KUKA KRL program: machina_kuka_driver.src, machina_kuka_driver.dat

--- machina_kuka_driver.src ---
&ACCESS RVP
&REL 53
&PARAM DISKPATH = KRC:\R1\Program\Arastoo\Driver
&PARAM TEMPLATE = C:\KRC\Roboter\Template\vorgabe
&PARAM EDITMASK = *
DEF machina_kuka_driver( )

;FOLD INI
;FOLD BCO INI
GLOBAL INTERRUPT DECL 3 WHEN $STOPMESS==TRUE DO IR_STOPM ( )
INTERRUPT ON 3
BAS (#INITMOV,0 )
;ENDFOLD (BCO INI)
;ENDFOLD (INI)



; For KUKA 3 files need to be installed: .src driver, .dat data file, and .xml server configurations
; in the xml file we specify the precise format of each action, accessed by the src driver program
; This file starts a TCP server on a real KUKA robot,
; waits for a TCP client, listens to a stream of formatted string messages in xml,
; buffers them parsed into an 'action' struct, and runs a loop to execute them.

; IMPORTANT: make sure to adjust {{HOSTNAME}} and {{PORT}} to your current setup
; More info on https://github.com/RobotExMachina
; A project by https://github.com/garciadelcastillo

; MIT License

; Copyright (c) 2018 Jose Luis Garcia del Castillo y Lopez

; Permission is hereby granted, free of charge, to any person obtaining a copy
; of this software and associated documentation files (the "Software"), to deal
; in the Software without restriction, including without limitation the rights
; to use, copy, modify, merge, publish, distribute, sublicense, and/or sell
; copies of the Software, and to permit persons to whom the Software is
; furnished to do so, subject to the following conditions:

; The above copyright notice and this permission notice shall be included in all
; copies or substantial portions of the Software.

; THE SOFTWARE IS PROVIDED "AS IS", WITHOUT WARRANTY OF ANY KIND, EXPRESS OR
; IMPLIED, INCLUDING BUT NOT LIMITED TO THE WARRANTIES OF MERCHANTABILITY,
; FITNESS FOR A PARTICULAR PURPOSE AND NONINFRINGEMENT. IN NO EVENT SHALL THE
; AUTHORS OR COPYRIGHT HOLDERS BE LIABLE FOR ANY CLAIM, DAMAGES OR OTHER
; LIABILITY, WHETHER IN AN ACTION OF CONTRACT, TORT OR OTHERWISE, ARISING FROM,
; OUT OF OR IN CONNECTION WITH THE SOFTWARE OR THE USE OR OTHER DEALINGS IN THE
; SOFTWARE.

; specifying the robot will read 3 commands in advance so that it can blend movements
$ADVANCE=3

; Initializing a TCP server on the robot and listening for clients and messages
RET=EKI_Init("machina_kuka_server")
RET=EKI_Open("machina_kuka_server")

;PTP {A1 0,A2 -85,A3 105,A4 0,A5 -20,A6 0}
;FOLD INI
;FOLD BCO INI
GLOBAL INTERRUPT DECL 3 WHEN $STOPMESS==TRUE DO IR_STOPM ( )
INTERRUPT ON 3
BAS (#INITMOV,0 )
;ENDFOLD (BCO INI)
;ENDFOLD (INI)

; Setting status and turn for the initial position of the robot
; status and turn define the joint configuration of a robot for a position
joint_pos_tgt = $axis_act_meas
PTP joint_pos_tgt
current_position = $POS_ACT_MES
IK_pose_position = {X 0,Y 0,Z 0,A 0,B 0,C 0}
IK_pose_position.X = current_position.X
IK_pose_position.Y = current_position.Y
IK_pose_position.Z = current_position.Z
IK_pose_position.A = current_position.A
IK_pose_position.B = current_position.B
IK_pose_position.C = current_position.C
PTP IK_pose_position C_PTP
$TOOL = $NULLFRAME

$VEL.CP=0.02
FOR FI=1 TO 6
$VEL_AXIS[FI] = 10 ;all axis velocities to 10%
ENDFOR

; setting default movement path blending values
$APO.CDIS = 5
$APO.CPTP = 5

wait for $FLAG[1] ;Please Connect Machina Bridge To the Robot!
$FLAG[32] = FALSE
IF $FLAG[1] == TRUE THEN

; get the current position of the robot to stream to machina bridge
current_axispos = $AXIS_ACT_MEAS
current_posmove = $POS_ACT_MES

;Read and send the current position data to Machina
RET = eki_setreal("machina_kuka_server", "S/@VR", driver_ver)
RET = eki_setreal("machina_kuka_server", "S/@A1", current_axispos.A1)
RET = eki_setreal("machina_kuka_server", "S/@A2", current_axispos.A2)
RET = eki_setreal("machina_kuka_server", "S/@A3", current_axispos.A3)
RET = eki_setreal("machina_kuka_server", "S/@A4", current_axispos.A4)
RET = eki_setreal("machina_kuka_server", "S/@A5", current_axispos.A5)
RET = eki_setreal("machina_kuka_server", "S/@A6", current_axispos.A6)
RET = eki_setreal("machina_kuka_server", "S/@X", current_posmove.X)
RET = eki_setreal("machina_kuka_server", "S/@Y", current_posmove.Y)
RET = eki_setreal("machina_kuka_server", "S/@Z", current_posmove.Z)
RET = eki_setreal("machina_kuka_server", "S/@A", current_posmove.A)
RET = eki_setreal("machina_kuka_server", "S/@B", current_posmove.B)
RET = eki_setreal("machina_kuka_server", "S/@C", current_posmove.C)

RET = eki_send("machina_kuka_server", "S")

ENDIF

;instantiation
FOR FI = 1 TO 200 STEP 1
actions[FI].id = -1
actions[FI].type = -1
actions[FI].v1 = -1000
actions[FI].v2 = -1000
actions[FI].v3 = -1000
actions[FI].v4 = -1000
actions[FI].v5 = -1000
actions[FI].v6 = -1000
actions[FI].v7 = -1000
actions[FI].msg[] = "place holder"
ENDFOR
MessagePath[] = "DT/Msg/Str/@M05"
pathextent1[] = "000000000111111"
pathextent2[] = "123456789012345"
act_message[] = "place holder"
msg_type = 0
action_motion_mode = 0 ;Default motion mode is linear
action_d_out_index = -1
action_d_out_state = 0 ;Default digital output is false

FOR FI = 1 TO 15 STEP 1
ids[FI] = -1
types[FI] = -1
newacts_v1[FI] = -1000
newacts_v2[FI] = -1000
newacts_v3[FI] = -1000
newacts_v4[FI] = -1000
newacts_v5[FI] = -1000
newacts_v6[FI] = -1000
newacts_v7[FI] = -1000
ENDFOR

;current = 1
lastaction = 0
;dataCount = 0


WAIT FOR $FLAG[2] ; Watinging For Actions!
read_data_cnn()
populate_lst()
$FLAG[2] = FALSE

;start of the infinite loop
LOOP

FOR FI = 1 TO 200 STEP 1

;Default Non-Action = -1
;Undefined = 00
;Translation = 01
;Rotation = 02
;Transformation = 03
;Axes = 04
;Message = 05
;Wait = 06
;Speed = 07
;Acceleration = 08
;Precision = 09
;MotionMode = 10
;Coordinates = 11
;PushPop = 12
;Comment = 13
;DefineTool = 14
;AttachTool = 15
;DetachTool = 16
;IODigital = 17
;IOAnalog = 18
;Temperature = 19
;Extrusion = 20
;ExtrusionRate = 21
;Initialization = 22
;ExternalAxis = 23
;CustomCode = 24
;ArmAngle = 25

; a switch case block that executes actions according to their types
SWITCH actions[FI].type

CASE -1,-2
startover = TRUE
IF startover == TRUE THEN
WAIT FOR $FLAG[2]
startover = FALSE
lastaction = 0
ENDIF

IF $FLAG[2] == TRUE THEN
read_data_cnn()
repopulate_lst()
$FLAG[2] = FALSE
ENDIF
; default non-action for breaking the for loop and going back to waiting for messasges
 EXIT

CASE 0 ;Undefined = 00
; Do Nothing

CASE 1 ;Translation = 01
 moveframe.X = actions[FI].v2
 moveframe.Y = actions[FI].v3
 moveframe.Z = actions[FI].v4
 IF actions[FI].v1 == 1 THEN
 PTP moveframe C_PTP
 ELSE
 LIN moveframe C_DIS
 ENDIF

CASE 2 ;Rotation = 02
 posmove.x = actions[FI].v2
 posmove.y = actions[FI].v3
 posmove.z = actions[FI].v4
 posmove.a = actions[FI].v5
 posmove.b = actions[FI].v6
 posmove.c = actions[FI].v7
 LIN posmove C_DIS

CASE 3 ;Transformation = 03
 posmove.x = actions[FI].v2
 posmove.y = actions[FI].v3
 posmove.z = actions[FI].v4
 posmove.a = actions[FI].v5
 posmove.b = actions[FI].v6
 posmove.c = actions[FI].v7

 IF actions[FI].v1 == 1 THEN
 PTP posmove C_PTP
 ELSE
 LIN posmove C_DIS
 ENDIF

CASE 4 ;Axes = 04
 axispos.A1 = actions[FI].v2
 axispos.A2 = actions[FI].v3
 axispos.A3 = actions[FI].v4
 axispos.A4 = actions[FI].v5
 axispos.A5 = actions[FI].v6
 axispos.A6 = actions[FI].v7
 PTP axispos C_PTP

CASE 5 ;Message = 05
   msg_type = actions[FI].v1
   SWITCH msg_type

     CASE 1
     ;Notification Interface
     Messenger = {Modul[] "machina_kuka_driver",Nr 1,Msg_txt[] "PlaceHolder"}
     Messenger.Msg_txt[] =  actions[FI].msg[]
     Messenger.NR = FI
     Parameter[1]= {Par_type #empty}
     Parameter[2]= {Par_type #empty}
     Parameter[3]= {Par_type #empty}
     Opt = {VL_Stop TRUE, Clear_P_Reset TRUE, Clear_P_SAW FALSE, Log_To_DB FALSE}
     Ticket = Set_KrlMsg (#Notify,Messenger,Parameter[],Opt)

     CASE 2
     ;Alert Interface
     Messenger = {Modul[] "machina_kuka_driver",Nr 1,Msg_txt[] "PlaceHolder"}
     Messenger.Msg_txt[] =  actions[FI].msg[]
     Messenger.NR = FI
     Parameter[1]= {Par_type #empty}
     Parameter[2]= {Par_type #empty}
     Parameter[3]= {Par_type #empty}
     Opt = {VL_Stop TRUE, Clear_P_Reset TRUE, Clear_P_SAW FALSE, Log_To_DB FALSE}
     Ticket = Set_KrlMsg (#Quit,Messenger,Parameter[],Opt)

     CASE 3
     ;Critical Alert Interface
     ;Alert Interface
     Messenger = {Modul[] "machina_kuka_driver",Nr 1,Msg_txt[] "PlaceHolder"}
     Messenger.Msg_txt[] =  actions[FI].msg[]
     Messenger.NR = FI
     Parameter[1]= {Par_type #empty}
     Parameter[2]= {Par_type #empty}
     Parameter[3]= {Par_type #empty}
     Opt = {VL_Stop TRUE, Clear_P_Reset TRUE, Clear_P_SAW FALSE, Log_To_DB FALSE}
     Ticket = Set_KrlMsg (#Quit,Messenger,Parameter[],Opt)
     HALT

     CASE 4
     ;State Interface
     Messenger = {Modul[] "machina_kuka_driver",Nr 1,Msg_txt[] "PlaceHolder"}
     Messenger.Msg_txt[] =  actions[FI].msg[]
     Messenger.NR = FI
     Parameter[1]= {Par_type #empty}
     Parameter[2]= {Par_type #empty}
     Parameter[3]= {Par_type #empty}
     Opt = {VL_Stop TRUE, Clear_P_Reset TRUE, Clear_P_SAW TRUE, Log_To_DB FALSE}
     Ticket = Set_KrlMsg (#State,Messenger,Parameter[],Opt)

     DEFAULT
     ; Do nothing
   ENDSWITCH

CASE 6 ;Wait = 06
 WAIT SEC actions[FI].v1

CASE 7 ;Speed = 07
 $VEL.CP = actions[FI].v1
 axisSpeed = actions[FI].v2
 FOR tempindex=1 TO 6
 $VEL_AXIS[tempindex] = axisSpeed ;all axis velocities to 10%
 ENDFOR

CASE 8 ;Acceleration = 08

CASE 9 ;Precision = 09
 $APO.CDIS = actions[FI].v1

;CASE 10 ;MotionMode = 10
; action_motion_mode = actions[FI].v1

CASE 11 ;Coordinates = 11

CASE 12 ;PushPop = 12

CASE 13 ;Comment = 13

CASE 14 ;DefineTool = 14
 ; tool name set
CASE 15 ;AttachTool = 15
 toolframe.x = actions[FI].v2
 toolframe.y = actions[FI].v3
 toolframe.z = actions[FI].v4
 toolframe.a = actions[FI].v5
 toolframe.b = actions[FI].v6
 toolframe.c = actions[FI].v7
 $TOOL = toolframe

CASE 16 ;DetachTool = 16
 $TOOL = $NULLFRAME

CASE 17 ;IODigital = 17
 action_d_out_index = actions[FI].v1
 action_d_out_state = actions[FI].v2
 IF action_d_out_state == 0 THEN

 CONTINUE
 TRIGGER WHEN DISTANCE=0 DELAY=0 DO $OUT[action_d_out_index] = FALSE
 ;$OUT[action_d_out_index] = FALSE
 ENDIF
 IF action_d_out_state == 1 THEN
 CONTINUE
 TRIGGER WHEN DISTANCE=0 DELAY=0 DO $OUT[action_d_out_index] = TRUE
 ;$OUT[action_d_out_index] = TRUE
 ENDIF

CASE 18 ;IOAnalog = 18

CASE 19 ;Temperature = 19

CASE 20 ;Extrusion = 20

CASE 21 ;ExtrusionRate = 21

CASE 22 ;Initialization = 22

CASE 23 ;ExternalAxis = 23

CASE 24 ;CustomCode = 24

CASE 25 ;ArmAngle = 25
 axispos.A1 = actions[FI].v2
 axispos.A2 = actions[FI].v3
 axispos.A3 = actions[FI].v4
 axispos.A4 = actions[FI].v5
 axispos.A5 = actions[FI].v6
 axispos.A6 = actions[FI].v7
 PTP axispos C_PTP

DEFAULT
; Do Nothing

ENDSWITCH


; right after executing an action we check if we have more incoming actions from Machina
IF $FLAG[2] == TRUE THEN
read_data_cnn()
repopulate_lst()
$FLAG[2] = FALSE
ENDIF

; after each action execution we send feedback to machina bridge
machinafeedback()
actions[FI].type = -1

ENDFOR

; end of the infinite loop
ENDLOOP

END

DEF machinafeedback( )

;Undefined = 00
;Translation = 01
;Rotation = 02
;Transformation = 03
;Axes = 04
;Message = 05
;Wait = 06
;Speed = 07
;Acceleration = 08
;Precision = 09
;MotionMode = 10
;Coordinates = 11
;PushPop = 12
;Comment = 13
;DefineTool = 14
;AttachTool = 15
;DetachTool = 16
;IODigital = 17
;IOAnalog = 18
;Temperature = 19
;Extrusion = 20
;ExtrusionRate = 21
;Initialization = 22
;ExternalAxis = 23
;CustomCode = 24
;ArmAngle = 25
IF actions[FI].type > -1 THEN

RET = eki_setint("machina_kuka_server", "R/@ID", actions[FI].id)
RET = eki_setint("machina_kuka_server", "R/@T", actions[FI].type)

; setting the flag 32 and making the robot wait for milliseconds creates
; enough time for feedback messages to be sent individually and to prevent
; message from merging
$FLAG[32] = TRUE
IF $FLAG[32] == TRUE THEN

SWITCH actions[FI].type
 ;Message = 05 Speed = 07 Acceleration = 08 Precision = 09 MotionMode = 10
 ;Comment = 13 DefineTool = 14 AttachTool = 15 IODigital = 17 IOAnalog = 18
 CASE 5,7,8,9,10,13,14,15,17,18
   continue
   WAIT SEC 0.2
 DEFAULT
   continue
   WAIT SEC 0.05

ENDSWITCH

; send feedback
RET = eki_send("machina_kuka_server", "R")
RET = EKI_ClearBuffer("machina_kuka_server", "R")
ENDIF

$FLAG[32] = FALSE

ENDIF

END
DEF read_data_cnn( )
;A function to read actions from the incomin stream
RET = eki_getint("machina_kuka_server", "DT/DC", newdatacount)
RET = eki_getintarray("machina_kuka_server", "DT/DR/A/@ID", ids[])
RET = eki_getintarray("machina_kuka_server", "DT/DR/A/@T", types[])
RET = eki_getrealarray("machina_kuka_server", "DT/DR/A/@V1", newacts_v1[])
RET = eki_getrealarray("machina_kuka_server", "DT/DR/A/@V2", newacts_v2[])
RET = eki_getrealarray("machina_kuka_server", "DT/DR/A/@V3", newacts_v3[])
RET = eki_getrealarray("machina_kuka_server", "DT/DR/A/@V4", newacts_v4[])
RET = eki_getrealarray("machina_kuka_server", "DT/DR/A/@V5", newacts_v5[])
RET = eki_getrealarray("machina_kuka_server", "DT/DR/A/@V6", newacts_v6[])
RET = eki_getrealarray("machina_kuka_server", "DT/DR/A/@V7", newacts_v7[])

END
DEF populate_lst( )
; A function to add incoming actions to the actions array
FOR popfi = 1 TO newdatacount STEP 1


index = popfi + lastaction
actions[index].ID = ids[popfi]
actions[index].type = types[popfi]
actions[index].v1 = newacts_v1[popfi]
actions[index].v2 = newacts_v2[popfi]
actions[index].v3 = newacts_v3[popfi]
actions[index].v4 = newacts_v4[popfi]
actions[index].v5 = newacts_v5[popfi]
actions[index].v6 = newacts_v6[popfi]
actions[index].v7 = newacts_v7[popfi]

IF types[popfi] == 5 THEN
MessagePath[14] = pathextent1[popfi]
MessagePath[15] = pathextent2[popfi]
RET = eki_getstring("machina_kuka_server", MessagePath[], act_message[])
actions[index].msg[] = act_message[]
ENDIF

ENDFOR

lastaction = lastaction + newdatacount

RET = EKI_ClearBuffer("machina_kuka_server", "DT")
END
DEF repopulate_lst( )
;A function to add incoming actions to the action array while the robot is moving
tempindex = 1

FOR repopfi = 1 TO newdatacount STEP 1

 index = repopfi + lastaction

; We have limited memory on the robot so we have to rewrite the action queue
 IF index > 200 THEN
 wrap = TRUE
 index = repopfi + lastaction - 200
 ENDIF

 actions[index].ID = ids[repopfi]
 actions[index].type = types[repopfi]
 actions[index].v1 = newacts_v1[repopfi]
 actions[index].v2 = newacts_v2[repopfi]
 actions[index].v3 = newacts_v3[repopfi]
 actions[index].v4 = newacts_v4[repopfi]
 actions[index].v5 = newacts_v5[repopfi]
 actions[index].v6 = newacts_v6[repopfi]
 actions[index].v7 = newacts_v7[repopfi]

 IF types[repopfi] == 5 THEN
 MessagePath[14] = pathextent1[repopfi]
 MessagePath[15] = pathextent2[repopfi]
 RET = eki_getstring("machina_kuka_server", MessagePath[], act_message[])
 actions[index].msg[] = act_message[]
 ENDIF

ENDFOR

IF wrap == FALSE THEN
lastaction = lastaction + newdatacount
ELSE
lastaction = index
wrap = FALSE
ENDIF
; clearning the TCP buffer prevents memory overload on the robot
RET = EKI_ClearBuffer("machina_kuka_server", "DT")
END

--- machina_kuka_driver.dat ---
&ACCESS RVP
&REL 53
&PARAM DISKPATH = KRC:\R1\Program\Arastoo\Driver
&PARAM TEMPLATE = C:\KRC\Roboter\Template\vorgabe
&PARAM EDITMASK = *
DEFDAT  machina_kuka_driver

; This file starts a synchronous, single-threaded server on a virtual/real ABB robot,
; waits for a TCP client, listens to a stream of formatted string messages,
; buffers them parsed into an 'action' struct, and runs a loop to execute them.

; IMPORTANT: make sure to adjust {{HOSTNAME}} and {{PORT}} to your current setup
; More info on https://github.com/RobotExMachina
; A project by https://github.com/garciadelcastillo

; MIT License

; Copyright (c) 2018 Jose Luis Garcia del Castillo y Lopez

; Permission is hereby granted, free of charge, to any person obtaining a copy
; of this software and associated documentation files (the "Software"), to deal
; in the Software without restriction, including without limitation the rights
; to use, copy, modify, merge, publish, distribute, sublicense, and/or sell
; copies of the Software, and to permit persons to whom the Software is
; furnished to do so, subject to the following conditions:

; The above copyright notice and this permission notice shall be included in all
; copies or substantial portions of the Software.

; THE SOFTWARE IS PROVIDED "AS IS", WITHOUT WARRANTY OF ANY KIND, EXPRESS OR
; IMPLIED, INCLUDING BUT NOT LIMITED TO THE WARRANTIES OF MERCHANTABILITY,
; FITNESS FOR A PARTICULAR PURPOSE AND NONINFRINGEMENT. IN NO EVENT SHALL THE
; AUTHORS OR COPYRIGHT HOLDERS BE LIABLE FOR ANY CLAIM, DAMAGES OR OTHER
; LIABILITY, WHETHER IN AN ACTION OF CONTRACT, TORT OR OTHERWISE, ARISING FROM,
; OUT OF OR IN CONNECTION WITH THE SOFTWARE OR THE USE OR OTHER DEALINGS IN THE
; SOFTWARE.

; For loop incrementing Integer Variables
DECL INT FI
DECL INT popfi
DECL INT repopfi
DECL INT readfi
; List aciton poplulation indecies
DECL REAL driver_ver=1.0
DECL INT lastaction=1
DECL INT current=2
DECL INT index=1
DECL INT tempindex=1
DECL INT dataCount=8
DECL INT newdatacount=1
DECL BOOL wrap=FALSE
DECL BOOL startover=TRUE
DECL INT axisSpeed=0

;BCO Variables
DECL AXIS joint_pos_tgt
DECL POS current_position
DECL POS IK_pose_position

; Messaging Interface variables
DECL EKI_STATUS RET
DECL CHAR MessagePath[15] ;path is used in the eki_getstring() function for the xml path finding
DECL CHAR pathextent1[15] ; for a string of numbers like "000000000111111" for searching for the path number char -> "0 "
DECL CHAR pathextent2[15] ; for a string of numbers like "123456789012345" for searching for the path number char -> " 5" --> "05"
DECL CHAR act_message[80] ; length of a messsage to be sent to the contorller is 80 characters
DECL KRLMSG_T Messenger
DECL KRLMSGPAR_T Parameter[3]
DECL KRLMSGOPT_T Opt
DECL INT Ticket
DECL INT msg_type
DECL INT action_motion_mode
DECL INT action_d_out_index
DECL INT action_d_out_state

; action properties
DECL INT actionType=-1
STRUC actionstruct INT id,INT type,REAL v1,REAL v2,REAL v3,REAL v4,REAL v5,REAL v6,REAL v7,CHAR msg[80] ; a struct for all the actions to be cast to
DECL actionstruct actions[200]
; arrays to receive data from the TCP buffer
DECL INT ids[15]
DECL INT types[15]
DECL REAL newacts_v1[15]
DECL REAL newacts_v2[15]
DECL REAL newacts_v3[15]
DECL REAL newacts_v4[15]
DECL REAL newacts_v5[15]
DECL REAL newacts_v6[15]
DECL REAL newacts_v7[15]

;motion position variables
POS posmove={X 1455.5,Y 123.0,Z 137.0,A 0.0,B 90.0,C 0.0,S 'B0010'}
AXIS axispos={A1 0.0,A2 -85.0,A3 105.0,A4 0.0,A5 -20.0,A6 0.0}
DECL FRAME moveframe={X 1122.75806,Y -318.985992,Z 833.369019}
DECL FRAME toolframe={X 234.621994,Y 2.7349999,Z 70.7060013,A 0.0,B 0.0,C 0.0}

;current position status
AXIS current_axispos={A1 -6.00493336,A2 -54.8471794,A3 90.9039688,A4 -190.071884,A5 36.6114769,A6 -171.896576}
POS current_sudoAxis={X 1060.0,Y -150.0,Z 1000.0,A 180.0,B 0.0,C 0.0}
POS current_posmove={X 1324.29065,Y 122.270988,Z 807.622925,A -86.7022171,B 89.9991837,C -86.7026062,S 'B00010010',T 'B00101011'}

ENDDAT
